(* IEC 61131-3 sources: AXOpen/src/messaging/ctrl/src/abstractions/IxMessage, 5 files *)

(* ---- IIxMessageProperties.st ---- *)
NAMESPACE ix.framework.messaging
    INTERFACE IIxMessageProperties
        METHOD Pin: IIxMessageProperties END_METHOD
        METHOD IsPinned: BOOL END_METHOD
    END_INTERFACE
END_NAMESPACE

(* ---- IIxMessages.st ---- *)
NAMESPACE ix.framework.core
    INTERFACE IIxMessages
	    /// <summary>
		/// Adds message of 'debug' category to the message queue.
		/// </summary>
        METHOD Debug : IIxMessageProperties
            VAR_INPUT
                /// <summary>
                /// Arbitrary message string.
                /// </summary>
                Message : STRING[IxIntConstants#MAX_MESSAGE_TEXT_LENGHT];
            END_VAR
        END_METHOD

	    /// <summary>
		/// Adds message of 'error' category to the message queue.
		/// </summary>
        METHOD Error : IIxMessageProperties
            VAR_INPUT
                /// <summary>
                /// Arbitrary message string.
                /// </summary>
                Message : STRING[IxIntConstants#MAX_MESSAGE_TEXT_LENGHT];
            END_VAR
        END_METHOD

	    /// <summary>
		/// Adds message of 'information' category to the message queue.
		/// </summary>
        METHOD Info : IIxMessageProperties
            VAR_INPUT
                /// <summary>
                /// Arbitrary message string.
                /// </summary>
                Message : STRING[IxIntConstants#MAX_MESSAGE_TEXT_LENGHT];
            END_VAR
        END_METHOD

	    /// <summary>
		/// Adds message of 'notification' category to the message queue.
		/// </summary>
        METHOD Notify : IIxMessageProperties
            VAR_INPUT
                /// <summary>
                /// Arbitrary message string.
                /// </summary>
                Message : STRING[IxIntConstants#MAX_MESSAGE_TEXT_LENGHT];
            END_VAR
        END_METHOD

	    /// <summary>
		/// Adds message of 'programming error' category to the message queue.
		/// </summary>
        METHOD Programming : IIxMessageProperties
            VAR_INPUT
                /// <summary>
                /// Arbitrary message string.
                /// </summary>
                Message : STRING[IxIntConstants#MAX_MESSAGE_TEXT_LENGHT];
            END_VAR
        END_METHOD

	    /// <summary>
		/// Adds message of 'trace' category to the message queue.
		/// </summary>
        METHOD Trace : IIxMessageProperties
            VAR_INPUT
                /// <summary>
                /// Arbitrary message string.
                /// </summary>
                Message : STRING[IxIntConstants#MAX_MESSAGE_TEXT_LENGHT];
            END_VAR
        END_METHOD

	    /// <summary>
		/// Adds message of 'warning' category to the message queue.
		/// </summary>
        METHOD Warning : IIxMessageProperties
            VAR_INPUT
                /// <summary>
                /// Arbitrary message string.
                /// </summary>
                Message : STRING[IxIntConstants#MAX_MESSAGE_TEXT_LENGHT];
            END_VAR
        END_METHOD

        METHOD Build: IIxMessageTextBuilder END_METHOD

        /// <summary>
		/// Adds message of given category to the message queue.
		/// </summary>
		/// <returns>Message index.</returns>
        METHOD Post  : IIxMessageProperties
            VAR_INPUT
                /// <summary>
                /// Arbitrary message string.
                /// </summary>
                Message : STRING[IxIntConstants#MAX_MESSAGE_TEXT_LENGHT];
                /// <summary>
                /// Message category.
                /// </summary>
                Category : eIxMessageCategory;
            END_VAR
        END_METHOD

		/// <summary>
		/// Unpins this messenger.
		/// </summary>
        METHOD UnPin END_METHOD

    END_INTERFACE
END_NAMESPACE

(* ---- IIxMessageTextBuilder.st ---- *)
NAMESPACE ix.framework.messaging
    INTERFACE IIxMessageTextBuilder
		/// <summary>
		/// Appends string to the message text.
		/// </summary>
		/// <remarks>
		/// 	<note type="warning">
		/// 		The size of the resulting string should not be more than '160' characters. The characters exceeding this size will be truncated.
		/// 	</note>
		/// </remarks>
        METHOD Append : IIxMessageTextBuilder
            VAR_INPUT
                Text : STRING[IxIntConstants#MAX_MESSAGE_TEXT_LENGHT];
            END_VAR
        END_METHOD

		/// <summary>
		/// Gets categorization methods for fluent message builder.
		/// </summary>
        METHOD As : IIxMessageCategorize END_METHOD

		/// <summary>
		/// Initiates new message text building for this messenger in fluent-like fashion.
		/// </summary>
        METHOD Build : IIxMessageTextBuilder END_METHOD
    END_INTERFACE
END_NAMESPACE

(* ---- IIxMessenger.st ---- *)
NAMESPACE ix.framework.core
    INTERFACE IIxMessenger
		/// <summary>
		/// Clears the message content.
		/// <remarks>
		/// 	<note type="important">
		/// 		This method is exposed for Rpc calls, for testing purposes. Rpc calls of this method must not be used in production code
		///		</note>
		/// </remarks>
		/// </summary>
		METHOD Clear END_METHOD

		METHOD OnCondition : IIxMessages
			VAR_INPUT
				inCondition : BOOL;
			END_VAR
		END_METHOD
    END_INTERFACE
END_NAMESPACE

(* ---- IIxMessengerEnv.st ---- *)
USING ix.framework.utils;

NAMESPACE ix.framework.messaging
    INTERFACE IIxMessengerEnv
		/// <summary>
		/// Gets whether the messaging is suspended at this point in program.
		/// <para>
		/// See also <see cref="PlcDocu.TcoCore.TcoMessengerSettings.Resume()"/>
		/// </para>
		/// <para>
		/// See also <see cref="PlcDocu.TcoCore.TcoMessengerSettings.Suspend()"/>
		/// </para>
		/// <para>
		/// See also <see cref="PlcDocu.TcoCore.TcoMessengerSettings.MinLevel"/>
		/// </para>
		/// </summary>
		METHOD IsSuspended: BOOL END_METHOD
		/// <summary>
		/// Gets the message digest method.
		/// Message digest serves to fingerprint messages.
		/// </summary>
		METHOD GetMessageDigestMethod : eIxMessageDigestMethod END_METHOD
		/// <summary>
		/// Sets the message digest method.
		/// Message digest serves to fingerprint messages.
		/// </summary>
		METHOD SetMessageDigestMethod VAR_INPUT inDigestMethod : eIxMessageDigestMethod; END_VAR END_METHOD
		/// <summary>
		/// Gets the minimal messaging level, the objects will post only messages for the levels of this or superior severity.
		/// <para>
		/// See also <see cref="PlcDocu.TcoCore.TcoMessengerSettings.Resume()"/>
		/// </para>
		/// <para>
		/// See also <see cref="PlcDocu.TcoCore.TcoMessengerSettings.Suspend()"/>
		/// </para>
		/// <para>
		/// See also <see cref="PlcDocu.TcoCore.TcoMessengerSettings.MinLevel"/>
		/// </para>
		/// </summary>
		METHOD GetMinLevel : eIxMessageCategory END_METHOD
		/// <summary>
		/// Sets the minimal messaging level, the objects will post only messages for the levels of this or superior severity.
		/// <para>
		/// See also <see cref="PlcDocu.TcoCore.TcoMessengerSettings.Resume()"/>
		/// </para>
		/// <para>
		/// See also <see cref="PlcDocu.TcoCore.TcoMessengerSettings.Suspend()"/>
		/// </para>
		/// <para>
		/// See also <see cref="PlcDocu.TcoCore.TcoMessengerSettings.MinLevel"/>
		/// </para>
		/// </summary>
		METHOD SetMinLevel VAR_INPUT inMessageCategory : eIxMessageCategory; END_VAR END_METHOD
		/// <summary>
		/// Resumes messaging from the all objects of this context, when the messaging was previously suspended by ```Suspend``` method.
		/// <para>
		/// See also <see cref="PlcDocu.TcoCore.TcoMessengerSettings.Suspend()"/>
		/// </para>
		/// <para>
		/// See also <see cref="PlcDocu.TcoCore.TcoMessengerSettings.MinLevel"/>
		/// </para>
		/// </summary>
		METHOD Resume END_METHOD
		/// <summary>
		/// Suspends messaging from the all objects of this context that would occur from this point in the call tree.
		/// <para>
		/// See also <see cref="PlcDocu.TcoCore.TcoMessengerSettings.Resume()"/>
		/// </para>
		/// <para>
		/// See also <see cref="PlcDocu.TcoCore.TcoMessengerSettings.MinLevel"/>
		/// </para>
		/// </summary>
		METHOD Suspend END_METHOD
		METHOD GetStringBuilder : REF_TO StringBuilder END_METHOD
	END_INTERFACE
END_NAMESPACE
